// TIA Portal project "IoT" (V15)

(* hardware
DEVICE "SIMATIC 315(r)"  S7-300 station
   slot 0: "Rack 0"  Rail  6ES7 390-1***0-0AA0
   slot 2: "CPU 315-2 PN/DP_1"  Unspecific CPU S7 300  6ES7 3XX-XXXXX-XXXX
DEVICE "SIMATIC 315(l)"  S7-300 station
   slot 0: "Rack 0"  Rail  6ES7 390-1***0-0AA0
   slot 2: "CPU 315-2 PN/DP"  Unspecific CPU S7 300  6ES7 3XX-XXXXX-XXXX
*)

// ===== PLC "CPU 315-2 PN/DP"  Unspecific CPU S7 300 =====

VAR_GLOBAL   // PLC tag table "STEP7 classic symbols"
   "TRUE" AT %M0.1 : Bool;
   "Startup" AT %M0.3 : Bool;
END_VAR

VAR_GLOBAL   // PLC tag table "Default tag table"
   "Tag_1" AT %M100.6 : Bool;
   "Tag_2" AT %M10.0 : Bool;
END_VAR

DATA_BLOCK "DB1"   // DB1
TITLE = Connection Parameters for TCON
{ S7_Optimized_Access := 'FALSE' }
AUTHOR : SIMATIC
FAMILY : COMM
NAME : TCON_PAR
VERSION : 0.1
   VAR
      OUCW_1 : Struct
         block_length : Word := WORD#16#0040;   // #!Connection_01!#
         id : Word := WORD#16#0001;
         connection_type : Byte := BYTE#16#12;
         active_est : Bool := TRUE;
         local_device_id : Byte := BYTE#16#02;
         local_tsap_id_len : Byte := BYTE#16#04;
         rem_subnet_id_len : Byte;
         rem_staddr_len : Byte := BYTE#16#04;
         rem_tsap_id_len : Byte := BYTE#16#04;
         next_staddr_len : Byte;
         local_tsap_id : Array[1..16] of Byte;
         rem_subnet_id : Array[1..6] of Byte;
         rem_staddr : Array[1..6] of Byte;
         rem_tsap_id : Array[1..16] of Byte;
         next_staddr : Array[1..6] of Byte;
         spare : Word;   // #!Connection_01!#
      END_STRUCT;
   END_VAR
BEGIN
   OUCW_1.local_tsap_id[1] := BYTE#16#49;
   OUCW_1.local_tsap_id[2] := BYTE#16#53;
   OUCW_1.local_tsap_id[3] := BYTE#16#4F;
   OUCW_1.local_tsap_id[4] := BYTE#16#31;
   OUCW_1.rem_staddr[1] := BYTE#16#C0;
   OUCW_1.rem_staddr[2] := BYTE#16#A8;
   OUCW_1.rem_staddr[4] := BYTE#16#1E;
   OUCW_1.rem_tsap_id[1] := BYTE#16#49;
   OUCW_1.rem_tsap_id[2] := BYTE#16#53;
   OUCW_1.rem_tsap_id[3] := BYTE#16#4F;
   OUCW_1.rem_tsap_id[4] := BYTE#16#31;
END_DATA_BLOCK

DATA_BLOCK "DB11"   // DB11
{ S7_Optimized_Access := 'FALSE' }
VERSION : 0.0
// stored: InstanceOfName FB1
"FB1"
BEGIN
END_DATA_BLOCK

DATA_BLOCK "SEND_DATA"   // DB100
{ S7_Optimized_Access := 'FALSE' }
VERSION : 0.1
   VAR
      SEND_DATA : Array[0..99] of Byte;   // vorläufige Platzhaltervariable
   END_VAR
BEGIN
END_DATA_BLOCK

DATA_BLOCK "RECV_DATA"   // DB200
{ S7_Optimized_Access := 'FALSE' }
VERSION : 0.1
   VAR
      RECV_DATA : Array[0..99] of Byte;   // vorläufige Platzhaltervariable
   END_VAR
BEGIN
END_DATA_BLOCK

FUNCTION_BLOCK "FB1"   // FB1, LAD
{ S7_Optimized_Access := 'FALSE' }
VERSION : 0.1
   VAR_INPUT
      INIT_COM : Bool;
      ABORT : Bool;
   END_VAR
   VAR
      CONNECTION_START : Bool;
      SR_CONN : Bool;
      CON_DONE : Bool;
      CON_ERROR : Bool;
      CON_BUSY : Bool;
      CON_STATUS : Word;
      CON_STATUS_SAVE : Word;
      SEND_REQ_P : Bool;
      SEND_REQ : Bool;
      SEND_DONE : Bool;
      SEND_BUSY : Bool;
      SEND_ERROR : Bool;
      SEND_STATUS : Word;
      SEND_STATUS_SAVE : Word;
      SR_SEND : Bool;
      RCV_NDR : Bool;
      RCV_BUSY : Bool;
      RCV_ERROR : Bool;
      RCV_STATUS : Word;
      RCV_STATUS_SAVE : Word;
      RCV_RLEN_SAVE : Int;
      RCV_RLEN : Int;
      SR_ABORT : Bool;
      ABORT_P : Bool;
      ABORT_BUSY : Bool;
      ABORT_DONE : Bool;
      ABORT_REQ : Bool;
      ABORT_ERROR : Bool;
      ABORT_STATUS : Word;
      ID : Word;
   END_VAR
   VAR_TEMP   // added for the SCL form of the ladder/FBD networks
      _w1 : Bool;
   END_VAR
BEGIN

REGION Network 1
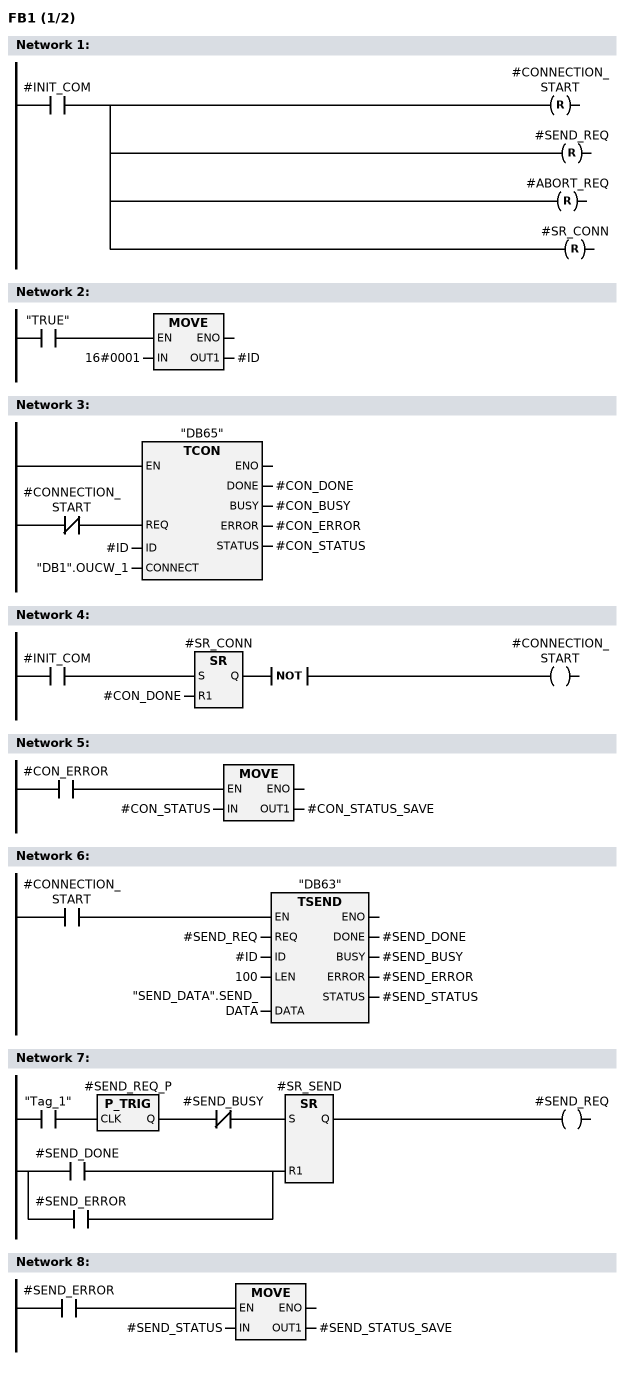
   RUNG wire#powerrail
      Contact( #INIT_COM )
      wire#w1
      R_Coil( #CONNECTION_START )
   END_RUNG
   RUNG wire#w1
      R_Coil( #SEND_REQ )
   END_RUNG
   RUNG wire#w1
      R_Coil( #ABORT_REQ )
   END_RUNG
   RUNG wire#w1
      R_Coil( #SR_CONN )
   END_RUNG
   // the same network as SCL:
   IF #INIT_COM THEN
       #CONNECTION_START := FALSE;
       #SEND_REQ := FALSE;
       #ABORT_REQ := FALSE;
       #SR_CONN := FALSE;
   END_IF;
END_REGION

REGION Network 2
   RUNG wire#powerrail
      Contact( "TRUE" )
      { S7_GenerateENO := "TRUE" } Move(in := 16#0001, out1 => #ID)
   END_RUNG
   // the same network as SCL:
   IF "TRUE" THEN #ID := 16#0001; END_IF;
END_REGION

REGION Network 3
   "DB65"(REQ := NOT #CONNECTION_START,   // TCON
          ID := #ID,
          CONNECT := "DB1".OUCW_1,
          DONE => #CON_DONE,
          BUSY => #CON_BUSY,
          ERROR => #CON_ERROR,
          STATUS => #CON_STATUS);
END_REGION

REGION Network 4
   RUNG wire#powerrail
      Contact( #INIT_COM )
      S_SR(operand := #SR_CONN, r1 := #CON_DONE)
      Not()
      Coil( #CONNECTION_START )
   END_RUNG
   // the same network as SCL:
   IF #INIT_COM THEN
       #SR_CONN := TRUE;   // SR flip-flop
   END_IF;
   IF #CON_DONE THEN #SR_CONN := FALSE; END_IF;
   #CONNECTION_START := NOT #SR_CONN;
END_REGION

REGION Network 5
   RUNG wire#powerrail
      Contact( #CON_ERROR )
      { S7_GenerateENO := "TRUE" } Move(in := #CON_STATUS, out1 => #CON_STATUS_SAVE)
   END_RUNG
   // the same network as SCL:
   IF #CON_ERROR THEN #CON_STATUS_SAVE := #CON_STATUS; END_IF;
END_REGION

REGION Network 6
   IF #CONNECTION_START THEN
       "DB63"(REQ := #SEND_REQ,   // TSEND
              ID := #ID,
              LEN := 100,
              DATA := "SEND_DATA".SEND_DATA,
              DONE => #SEND_DONE,
              BUSY => #SEND_BUSY,
              ERROR => #SEND_ERROR,
              STATUS => #SEND_STATUS);
   END_IF;
END_REGION

REGION Network 7
   RUNG wire#powerrail
      Contact( "Tag_1" )
      P_Trig( #SEND_REQ_P )
      I_Contact( #SEND_BUSY )
      S_SR(operand := #SR_SEND, r1 := wire#w1)
      Coil( #SEND_REQ )
   END_RUNG
   RUNG wire#powerrail
      Contact( #SEND_DONE )
   END_RUNG wire#w1
   RUNG wire#powerrail
      Contact( #SEND_ERROR )
   END_RUNG wire#w1
   // the same network as SCL:
   #_w1 := "Tag_1" AND NOT #SEND_REQ_P;   // rising edge
   #SEND_REQ_P := "Tag_1";
   IF #_w1 AND NOT #SEND_BUSY THEN
       #SR_SEND := TRUE;   // SR flip-flop
   END_IF;
   IF #SEND_DONE OR #SEND_ERROR THEN #SR_SEND := FALSE; END_IF;
   #SEND_REQ := #SR_SEND;
END_REGION

REGION Network 8
   RUNG wire#powerrail
      Contact( #SEND_ERROR )
      { S7_GenerateENO := "TRUE" } Move(in := #SEND_STATUS, out1 => #SEND_STATUS_SAVE)
   END_RUNG
   // the same network as SCL:
   IF #SEND_ERROR THEN #SEND_STATUS_SAVE := #SEND_STATUS; END_IF;
END_REGION

REGION Network 9
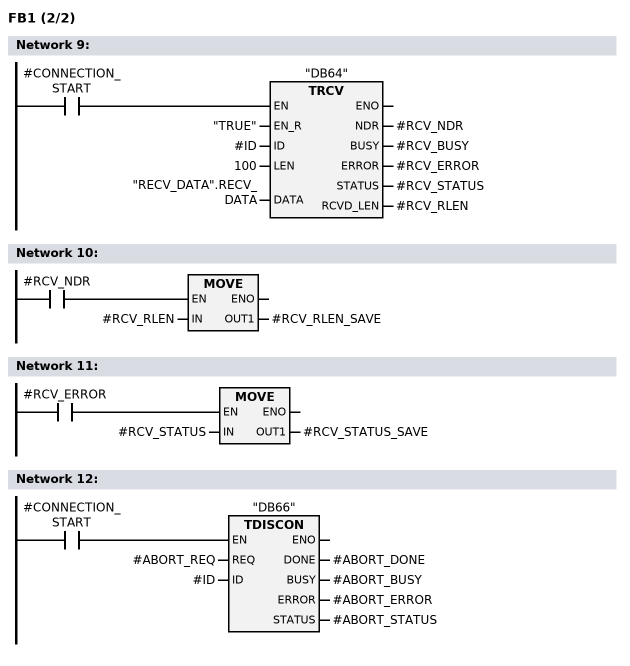
   IF #CONNECTION_START THEN
       "DB64"(EN_R := "TRUE",   // TRCV
              ID := #ID,
              LEN := 100,
              DATA := "RECV_DATA".RECV_DATA,
              NDR => #RCV_NDR,
              BUSY => #RCV_BUSY,
              ERROR => #RCV_ERROR,
              STATUS => #RCV_STATUS,
              RCVD_LEN => #RCV_RLEN);
   END_IF;
END_REGION

REGION Network 10
   RUNG wire#powerrail
      Contact( #RCV_NDR )
      { S7_GenerateENO := "TRUE" } Move(in := #RCV_RLEN, out1 => #RCV_RLEN_SAVE)
   END_RUNG
   // the same network as SCL:
   IF #RCV_NDR THEN #RCV_RLEN_SAVE := #RCV_RLEN; END_IF;
END_REGION

REGION Network 11
   RUNG wire#powerrail
      Contact( #RCV_ERROR )
      { S7_GenerateENO := "TRUE" } Move(in := #RCV_STATUS, out1 => #RCV_STATUS_SAVE)
   END_RUNG
   // the same network as SCL:
   IF #RCV_ERROR THEN #RCV_STATUS_SAVE := #RCV_STATUS; END_IF;
END_REGION

REGION Network 12
   IF #CONNECTION_START THEN
       "DB66"(REQ := #ABORT_REQ,   // TDISCON
              ID := #ID,
              DONE => #ABORT_DONE,
              BUSY => #ABORT_BUSY,
              ERROR => #ABORT_ERROR,
              STATUS => #ABORT_STATUS);
   END_IF;
END_REGION

REGION Network 13 (FBD)
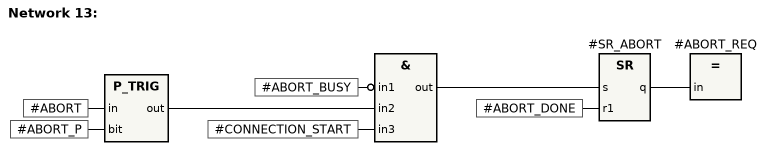
   #_w1 := #ABORT AND NOT #ABORT_P;   // rising edge
   #ABORT_P := #ABORT;
   IF NOT #ABORT_BUSY AND #_w1 AND #CONNECTION_START THEN
       #SR_ABORT := TRUE;   // SR flip-flop
   END_IF;
   IF #ABORT_DONE THEN #SR_ABORT := FALSE; END_IF;
   #ABORT_REQ := #SR_ABORT;
END_REGION
END_FUNCTION_BLOCK

ORGANIZATION_BLOCK "OB1"   // OB1, LAD
TITLE = "Main Program Sweep (Cycle)"
{ S7_Optimized_Access := 'FALSE' }
VERSION : 0.1
   VAR_TEMP
      OB1_EV_CLASS : Byte;   // Bits 0-3 = 1 (Coming event), Bits 4-7 = 1 (Event class 1)
      OB1_SCAN_1 : Byte;   // 1 (Cold restart scan 1 of OB 1), 3 (Scan 2-n of OB 1)
      OB1_PRIORITY : Byte;   // Priority of OB Execution
      OB1_OB_NUMBR : Byte;   // 1 (Organization block 1, OB1)
      OB1_RESERVED_1 : Byte;   // Reserved for system
      OB1_RESERVED_2 : Byte;   // Reserved for system
      OB1_PREV_CYCLE : Int;   // Cycle time of previous OB1 scan (milliseconds)
      OB1_MIN_CYCLE : Int;   // Minimum cycle time of OB1 (milliseconds)
      OB1_MAX_CYCLE : Int;   // Maximum cycle time of OB1 (milliseconds)
      OB1_DATE_TIME : Date_And_Time;   // Date and time OB1 started
   END_VAR
BEGIN

REGION Network 1
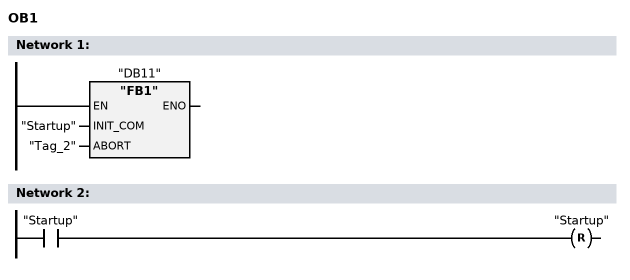
   RUNG wire#powerrail
      "DB11"(INIT_COM := "Startup", ABORT := "Tag_2")
   END_RUNG
   // the same network as SCL:
   "DB11"(INIT_COM := "Startup", ABORT := "Tag_2");   // "FB1"
END_REGION

REGION Network 2
   RUNG wire#powerrail
      Contact( "Startup" )
      R_Coil( "Startup" )
   END_RUNG
   // the same network as SCL:
   IF "Startup" THEN "Startup" := FALSE; END_IF;
END_REGION
END_ORGANIZATION_BLOCK

ORGANIZATION_BLOCK "COMPLETE RESTART"   // OB100, FBD
TITLE = "Complete Restart"
{ S7_Optimized_Access := 'FALSE' }
VERSION : 0.1
   VAR_TEMP
      OB100_EV_CLASS : Byte;   // 16#13, Event class 1, Entering event state, Event logged in diagnostic buffer
      OB100_STRTUP : Byte;   // 16#81/82/83/84 Method of startup
      OB100_PRIORITY : Byte;   // Priority of OB Execution
      OB100_OB_NUMBR : Byte;   // 100 (Organization block 100, OB100)
      OB100_RESERVED_1 : Byte;   // Reserved for system
      OB100_RESERVED_2 : Byte;   // Reserved for system
      OB100_STOP : Word;   // Event that caused CPU to stop (16#4xxx)
      OB100_STRT_INFO : DWord;   // Information on how system started
      OB100_DATE_TIME : Date_And_Time;   // Date and time OB100 started
   END_VAR
BEGIN

REGION Network 1
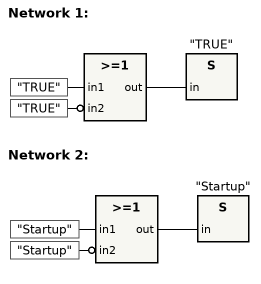
   IF "TRUE" OR NOT "TRUE" THEN "TRUE" := TRUE; END_IF;
END_REGION

REGION Network 2
   IF "Startup" OR NOT "Startup" THEN "Startup" := TRUE; END_IF;
END_REGION
END_ORGANIZATION_BLOCK

// ===== PLC "CPU 315-2 PN/DP_1"  Unspecific CPU S7 300 =====

VAR_GLOBAL   // PLC tag table "STEP7 classic symbols"
   "Startup" AT %M0.3 : Bool;
   "TRUE" AT %M0.1 : Bool;
END_VAR

VAR_GLOBAL   // PLC tag table "Default tag table"
   "Tag_1" AT %M100.6 : Bool;
   "Tag_2" AT %M10.0 : Bool;
END_VAR

DATA_BLOCK "DB1"   // DB1
TITLE = Connection Parameters for TCON
{ S7_Optimized_Access := 'FALSE' }
AUTHOR : SIMATIC
FAMILY : COMM
NAME : TCON_PAR
VERSION : 0.1
   VAR
      OUCW_1 : Struct
         block_length : Word := WORD#16#0040;   // #!Connection_01!#
         id : Word := WORD#16#0001;
         connection_type : Byte := BYTE#16#12;
         active_est : Bool;
         local_device_id : Byte := BYTE#16#02;
         local_tsap_id_len : Byte := BYTE#16#04;
         rem_subnet_id_len : Byte;
         rem_staddr_len : Byte := BYTE#16#04;
         rem_tsap_id_len : Byte := BYTE#16#04;
         next_staddr_len : Byte;
         local_tsap_id : Array[1..16] of Byte;
         rem_subnet_id : Array[1..6] of Byte;
         rem_staddr : Array[1..6] of Byte;
         rem_tsap_id : Array[1..16] of Byte;
         next_staddr : Array[1..6] of Byte;
         spare : Word;   // #!Connection_01!#
      END_STRUCT;
   END_VAR
BEGIN
   OUCW_1.local_tsap_id[1] := BYTE#16#49;
   OUCW_1.local_tsap_id[2] := BYTE#16#53;
   OUCW_1.local_tsap_id[3] := BYTE#16#4F;
   OUCW_1.local_tsap_id[4] := BYTE#16#31;
   OUCW_1.rem_staddr[1] := BYTE#16#C0;
   OUCW_1.rem_staddr[2] := BYTE#16#A8;
   OUCW_1.rem_staddr[4] := BYTE#16#14;
   OUCW_1.rem_tsap_id[1] := BYTE#16#49;
   OUCW_1.rem_tsap_id[2] := BYTE#16#53;
   OUCW_1.rem_tsap_id[3] := BYTE#16#4F;
   OUCW_1.rem_tsap_id[4] := BYTE#16#31;
END_DATA_BLOCK

DATA_BLOCK "DB11"   // DB11
{ S7_Optimized_Access := 'FALSE' }
VERSION : 0.0
// stored: InstanceOfName FB1
"FB1"
BEGIN
END_DATA_BLOCK

DATA_BLOCK "SEND_DATA"   // DB100
{ S7_Optimized_Access := 'FALSE' }
VERSION : 0.1
   VAR
      SEND_DATA : Array[0..99] of Byte;   // vorläufige Platzhaltervariable
   END_VAR
BEGIN
END_DATA_BLOCK

DATA_BLOCK "RECV_DATA"   // DB200
{ S7_Optimized_Access := 'FALSE' }
VERSION : 0.1
   VAR
      RECV_DATA : Array[0..99] of Byte;   // vorläufige Platzhaltervariable
   END_VAR
BEGIN
END_DATA_BLOCK

FUNCTION_BLOCK "FB1"   // FB1, LAD
{ S7_Optimized_Access := 'FALSE' }
VERSION : 0.1
   VAR_INPUT
      INIT_COM : Bool;
      ABORT : Bool;
   END_VAR
   VAR
      COMMUNICATION_START : Bool;
      CON_DONE : Bool;
      CON_BUSY : Bool;
      CON_ERROR : Bool;
      CON_STATUS : Word;
      CON_STATUS_SAVE : Word;
      SR_CON : Bool;
      SEND_REQ_P : Bool;
      SEND_REQ : Bool;
      SEND_DONE : Bool;
      SEND_BUSY : Bool;
      SEND_ERROR : Bool;
      SEND_STATUS : Word;
      SEND_STATUS_SAVE : Word;
      SR_SEND : Bool;
      RCV_NDR : Bool;
      RCV_BUSY : Bool;
      RCV_ERROR : Bool;
      RCV_STATUS : Word;
      RCV_STATUS_SAVE : Word;
      RCV_RLEN : Int;
      RCV_RLEN_SAVE : Int;
      ABORT_REQ : Bool;
      DIS_DONE : Bool;
      DIS_BUSY : Bool;
      DIS_ERROR : Bool;
      DIS_STATUS : Word;
      SR_ABORT : Bool;
      ABORT_REQ_P : Bool;
      ID : Word;
   END_VAR
   VAR_TEMP   // added for the SCL form of the ladder/FBD networks
      _w1 : Bool;
   END_VAR
BEGIN

REGION Network 1
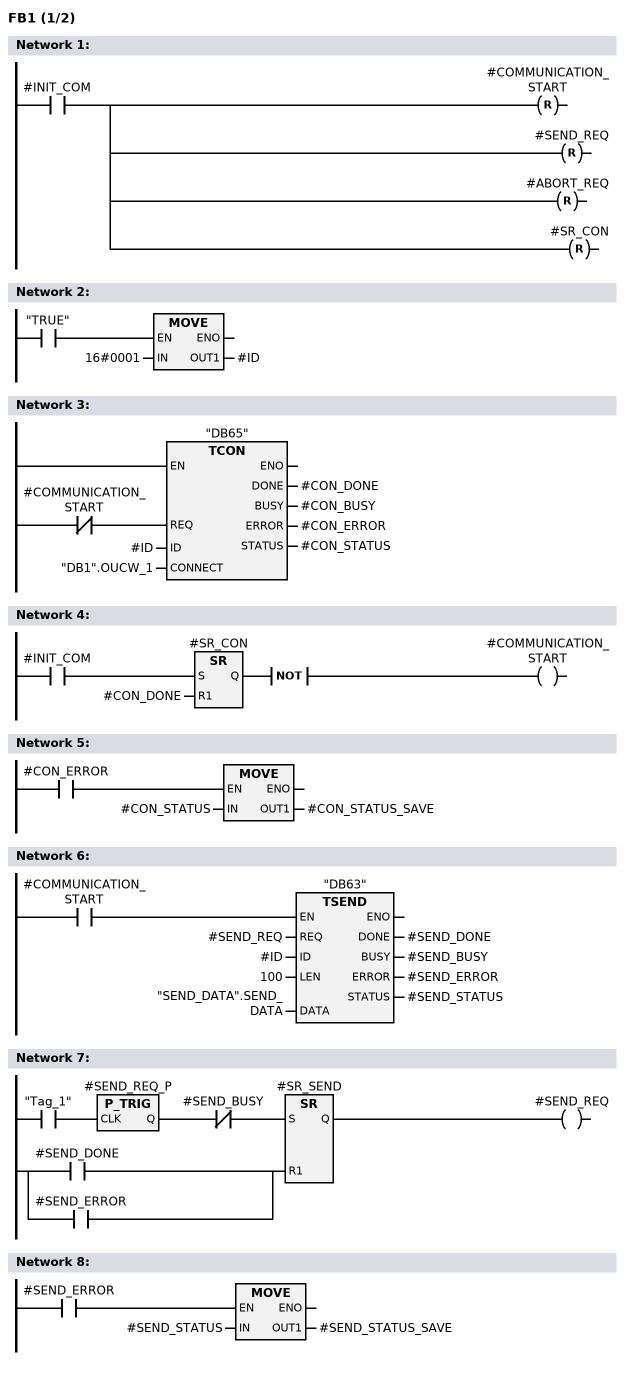
   RUNG wire#powerrail
      Contact( #INIT_COM )
      wire#w1
      R_Coil( #COMMUNICATION_START )
   END_RUNG
   RUNG wire#w1
      R_Coil( #SEND_REQ )
   END_RUNG
   RUNG wire#w1
      R_Coil( #ABORT_REQ )
   END_RUNG
   RUNG wire#w1
      R_Coil( #SR_CON )
   END_RUNG
   // the same network as SCL:
   IF #INIT_COM THEN
       #COMMUNICATION_START := FALSE;
       #SEND_REQ := FALSE;
       #ABORT_REQ := FALSE;
       #SR_CON := FALSE;
   END_IF;
END_REGION

REGION Network 2
   RUNG wire#powerrail
      Contact( "TRUE" )
      { S7_GenerateENO := "TRUE" } Move(in := 16#0001, out1 => #ID)
   END_RUNG
   // the same network as SCL:
   IF "TRUE" THEN #ID := 16#0001; END_IF;
END_REGION

REGION Network 3
   "DB65"(REQ := NOT #COMMUNICATION_START,   // TCON
          ID := #ID,
          CONNECT := "DB1".OUCW_1,
          DONE => #CON_DONE,
          BUSY => #CON_BUSY,
          ERROR => #CON_ERROR,
          STATUS => #CON_STATUS);
END_REGION

REGION Network 4
   RUNG wire#powerrail
      Contact( #INIT_COM )
      S_SR(operand := #SR_CON, r1 := #CON_DONE)
      Not()
      Coil( #COMMUNICATION_START )
   END_RUNG
   // the same network as SCL:
   IF #INIT_COM THEN
       #SR_CON := TRUE;   // SR flip-flop
   END_IF;
   IF #CON_DONE THEN #SR_CON := FALSE; END_IF;
   #COMMUNICATION_START := NOT #SR_CON;
END_REGION

REGION Network 5
   RUNG wire#powerrail
      Contact( #CON_ERROR )
      { S7_GenerateENO := "TRUE" } Move(in := #CON_STATUS, out1 => #CON_STATUS_SAVE)
   END_RUNG
   // the same network as SCL:
   IF #CON_ERROR THEN #CON_STATUS_SAVE := #CON_STATUS; END_IF;
END_REGION

REGION Network 6
   IF #COMMUNICATION_START THEN
       "DB63"(REQ := #SEND_REQ,   // TSEND
              ID := #ID,
              LEN := 100,
              DATA := "SEND_DATA".SEND_DATA,
              DONE => #SEND_DONE,
              BUSY => #SEND_BUSY,
              ERROR => #SEND_ERROR,
              STATUS => #SEND_STATUS);
   END_IF;
END_REGION

REGION Network 7
   RUNG wire#powerrail
      Contact( "Tag_1" )
      P_Trig( #SEND_REQ_P )
      I_Contact( #SEND_BUSY )
      S_SR(operand := #SR_SEND, r1 := wire#w1)
      Coil( #SEND_REQ )
   END_RUNG
   RUNG wire#powerrail
      Contact( #SEND_DONE )
   END_RUNG wire#w1
   RUNG wire#powerrail
      Contact( #SEND_ERROR )
   END_RUNG wire#w1
   // the same network as SCL:
   #_w1 := "Tag_1" AND NOT #SEND_REQ_P;   // rising edge
   #SEND_REQ_P := "Tag_1";
   IF #_w1 AND NOT #SEND_BUSY THEN
       #SR_SEND := TRUE;   // SR flip-flop
   END_IF;
   IF #SEND_DONE OR #SEND_ERROR THEN #SR_SEND := FALSE; END_IF;
   #SEND_REQ := #SR_SEND;
END_REGION

REGION Network 8
   RUNG wire#powerrail
      Contact( #SEND_ERROR )
      { S7_GenerateENO := "TRUE" } Move(in := #SEND_STATUS, out1 => #SEND_STATUS_SAVE)
   END_RUNG
   // the same network as SCL:
   IF #SEND_ERROR THEN #SEND_STATUS_SAVE := #SEND_STATUS; END_IF;
END_REGION

REGION Network 9
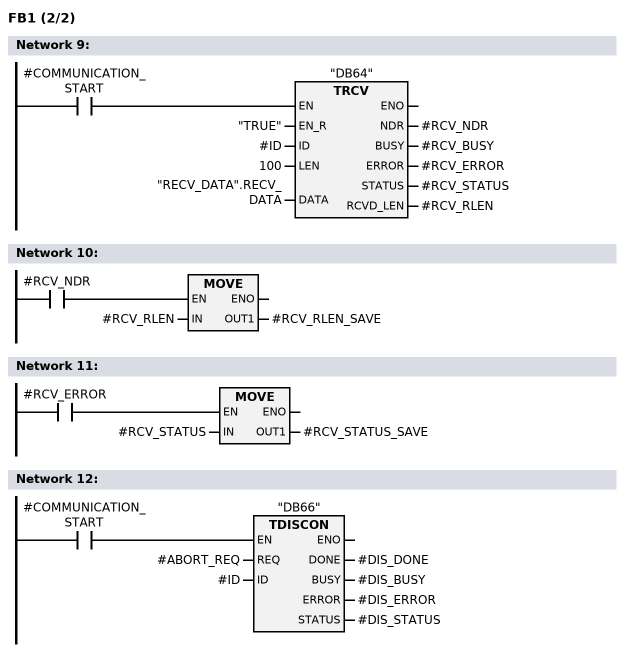
   IF #COMMUNICATION_START THEN
       "DB64"(EN_R := "TRUE",   // TRCV
              ID := #ID,
              LEN := 100,
              DATA := "RECV_DATA".RECV_DATA,
              NDR => #RCV_NDR,
              BUSY => #RCV_BUSY,
              ERROR => #RCV_ERROR,
              STATUS => #RCV_STATUS,
              RCVD_LEN => #RCV_RLEN);
   END_IF;
END_REGION

REGION Network 10
   RUNG wire#powerrail
      Contact( #RCV_NDR )
      { S7_GenerateENO := "TRUE" } Move(in := #RCV_RLEN, out1 => #RCV_RLEN_SAVE)
   END_RUNG
   // the same network as SCL:
   IF #RCV_NDR THEN #RCV_RLEN_SAVE := #RCV_RLEN; END_IF;
END_REGION

REGION Network 11
   RUNG wire#powerrail
      Contact( #RCV_ERROR )
      { S7_GenerateENO := "TRUE" } Move(in := #RCV_STATUS, out1 => #RCV_STATUS_SAVE)
   END_RUNG
   // the same network as SCL:
   IF #RCV_ERROR THEN #RCV_STATUS_SAVE := #RCV_STATUS; END_IF;
END_REGION

REGION Network 12
   IF #COMMUNICATION_START THEN
       "DB66"(REQ := #ABORT_REQ,   // TDISCON
              ID := #ID,
              DONE => #DIS_DONE,
              BUSY => #DIS_BUSY,
              ERROR => #DIS_ERROR,
              STATUS => #DIS_STATUS);
   END_IF;
END_REGION

REGION Network 13 (FBD)
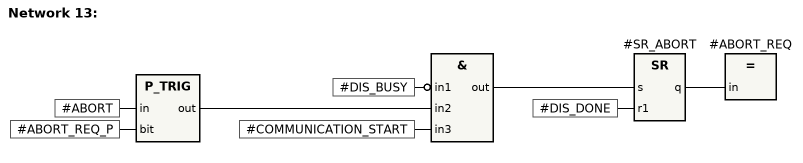
   #_w1 := #ABORT AND NOT #ABORT_REQ_P;   // rising edge
   #ABORT_REQ_P := #ABORT;
   IF NOT #DIS_BUSY AND #_w1 AND #COMMUNICATION_START THEN
       #SR_ABORT := TRUE;   // SR flip-flop
   END_IF;
   IF #DIS_DONE THEN #SR_ABORT := FALSE; END_IF;
   #ABORT_REQ := #SR_ABORT;
END_REGION
END_FUNCTION_BLOCK

ORGANIZATION_BLOCK "OB1"   // OB1, LAD
TITLE = "Main Program Sweep (Cycle)"
{ S7_Optimized_Access := 'FALSE' }
VERSION : 0.1
   VAR_TEMP
      OB1_EV_CLASS : Byte;   // Bits 0-3 = 1 (Coming event), Bits 4-7 = 1 (Event class 1)
      OB1_SCAN_1 : Byte;   // 1 (Cold restart scan 1 of OB 1), 3 (Scan 2-n of OB 1)
      OB1_PRIORITY : Byte;   // Priority of OB Execution
      OB1_OB_NUMBR : Byte;   // 1 (Organization block 1, OB1)
      OB1_RESERVED_1 : Byte;   // Reserved for system
      OB1_RESERVED_2 : Byte;   // Reserved for system
      OB1_PREV_CYCLE : Int;   // Cycle time of previous OB1 scan (milliseconds)
      OB1_MIN_CYCLE : Int;   // Minimum cycle time of OB1 (milliseconds)
      OB1_MAX_CYCLE : Int;   // Maximum cycle time of OB1 (milliseconds)
      OB1_DATE_TIME : Date_And_Time;   // Date and time OB1 started
   END_VAR
BEGIN

REGION Network 1
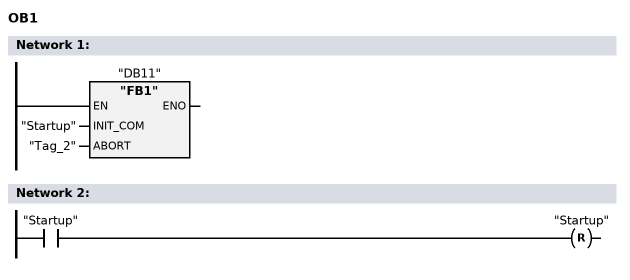
   RUNG wire#powerrail
      "DB11"(INIT_COM := "Startup", ABORT := "Tag_2")
   END_RUNG
   // the same network as SCL:
   "DB11"(INIT_COM := "Startup", ABORT := "Tag_2");   // "FB1"
END_REGION

REGION Network 2
   RUNG wire#powerrail
      Contact( "Startup" )
      R_Coil( "Startup" )
   END_RUNG
   // the same network as SCL:
   IF "Startup" THEN "Startup" := FALSE; END_IF;
END_REGION
END_ORGANIZATION_BLOCK

ORGANIZATION_BLOCK "COMPLETE RESTART"   // OB100, FBD
TITLE = "Complete Restart"
{ S7_Optimized_Access := 'FALSE' }
VERSION : 0.1
   VAR_TEMP
      OB100_EV_CLASS : Byte;   // 16#13, Event class 1, Entering event state, Event logged in diagnostic buffer
      OB100_STRTUP : Byte;   // 16#81/82/83/84 Method of startup
      OB100_PRIORITY : Byte;   // Priority of OB Execution
      OB100_OB_NUMBR : Byte;   // 100 (Organization block 100, OB100)
      OB100_RESERVED_1 : Byte;   // Reserved for system
      OB100_RESERVED_2 : Byte;   // Reserved for system
      OB100_STOP : Word;   // Event that caused CPU to stop (16#4xxx)
      OB100_STRT_INFO : DWord;   // Information on how system started
      OB100_DATE_TIME : Date_And_Time;   // Date and time OB100 started
   END_VAR
BEGIN

REGION Network 1
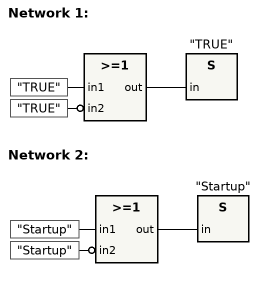
   IF "TRUE" OR NOT "TRUE" THEN "TRUE" := TRUE; END_IF;
END_REGION

REGION Network 2
   IF "Startup" OR NOT "Startup" THEN "Startup" := TRUE; END_IF;
END_REGION
END_ORGANIZATION_BLOCK